FUNCTION_BLOCK Test_TStreamAdd_Read_DINT_CheckAlignment EXTENDS T_UnitTestBase
VAR
    Stream  : T_Stream(StreamLength := 2);
    ArgType : E_ArgTypeId := E_ArgTypeId.Type_DINT;
END_VAR

METHOD  Init
VAR_INPUT
END_VAR
END_METHOD

{attribute 'analysis' := '-33'} // inhibit unused variable warning
METHOD RunTest
Stream.Init(2);

Stream.Add_BYTE(123);// add a byte to test alignment checks...
Stream.Add_DINT(12345678);

Stream.SetReadPosition(0);

Stream.Read_BYTE();

// check next value...	
AssertEquals_DINT(Expected     := 12345678,
                            Actual       := Stream.Read_DINT(),
                            Message := 'Stream.Read_DINT()');

// check we are at the end of the stream..							
AssertEquals_UDINT(Expected     := Stream.StreamLength,
                             Actual       := Stream.ReadPosition,
                             Message := 'Stream.ReadPosition');

TestCompleted := TRUE;
END_METHOD

END_FUNCTION_BLOCK

(* stored: Version 1.1.0.1, ProductVersion 3.1.4024.12
   POU Test_TStreamAdd_Read_DINT_CheckAlignment: Id {b15411b7-e134-45c3-9a68-12555b563d56}, SpecialFunc None
   Method Init: Id {b13ffd34-b1e0-46dd-a252-5bac8b77178f}
   Method RunTest: Id {e538cc6a-16e5-47e2-92fe-d84202776573} *)
